FUNCTION_BLOCK PlantNo2
VAR_INPUT
	lrInput : LREAL := 0.0;	
	
	lrM : LREAL := 4.72;
	lrC : LREAL := 2.9657;
	
	
END_VAR

VAR_OUTPUT
	lrOutput : LREAL := 0.0;
END_VAR

VAR
	arAccelerationHistory : ARRAY[0..5] OF LREAL := [0.0, 0.0, 0, 0, 0, 0];
	arVeloHistory : ARRAY[0..5] OF LREAL := [0.0, 0.0, 0, 0, 0, 0];
	arPositionHistory : ARRAY[0..5] OF LREAL := [0.0, 0.0, 0, 0, 0, 0];
	nCounter : INT := 0;

	lrTs : LREAL := 0.001;
END_VAR



FOR nCounter := 0 TO 4 DO
	arPositionHistory [5 - nCounter] := arPositionHistory[ 5 - nCounter -1];
	arVeloHistory [5 - nCounter] := arVeloHistory[ 5 - nCounter -1];
	arAccelerationHistory [5 - nCounter] := arAccelerationHistory[ 5 - nCounter -1];
END_FOR


arAccelerationHistory[0] := lrInput / lrM - lrC * arVeloHistory[0] / lrM;

arVeloHistory[0] := arVeloHistory[0] + 0.5 * lrTs * (arAccelerationHistory[0]+arAccelerationHistory[1]);

arPositionHistory[0] := arPositionHistory[0] + 0.5 * lrTs * (arVeloHistory[0]+arVeloHistory[1]);

lrOutput := arPositionHistory[0];

END_FUNCTION_BLOCK

(* stored: Version 1.1.0.1, ProductVersion 3.1.4026.8
   POU PlantNo2: Id {f6f3a758-0fca-4012-ae53-b14f819c7514}, SpecialFunc None *)
